PROGRAM OP70_CONVEYOR
VAR
	con_step_no : INT;
	cam_trig : BOOL;
	cam_ok : BOOL;
	LH_Cam_OK : BOOL;
	RH_Cam_OK : BOOL;
	t1: ton;
	t2: ton;
	t3: ton;
	t4: ton;
	
	temp: BOOL;
	check:BOOL;
	check1:ton;
	fwd_time : INT :=500;
	rev_time : INT :=500;	
	count_nok :INT;
	forward: BOOL;
	reverse: BOOL;

	temp1: BOOL;
	temp2: BOOL;
	
	LH_Cyl_Delay : TON;
	RH_Cyl_Delay : TON;
	temp_3: BOOL;
END_VAR

IF (NOT OP70_AutoSelected OR OP70_ErrorActive ) THEN
	//SR70_CONV_servo_ctrl.VELmove_Start:=FALSE;
	forward:=FALSE;
	reverse:=FALSE;
	con_step_no:= 10;
END_IF	



IF MANUAL_SELECTED AND OP70_ManualSelected THEN               
	IF I70_DRUM_CONV_REV_I308_3 THEN
		SR70_Conv_servo_status.targetVelocity:=OP70_Conv_Rev_Speed_6_3;
		SR70_CONV_servo_ctrl.VELmove_Start:=I70_DRUM_CONV_REV_I308_3;
 	ELSIF I70_DRUM_CONV_FWD_I308_4 THEN
		SR70_Conv_servo_status.targetVelocity:=OP70_Conv_Fwd_Speed_7_89;
		SR70_CONV_servo_ctrl.VELmove_Start:=I70_DRUM_CONV_FWD_I308_4;	
	ELSE 	
		SR70_CONV_servo_ctrl.VELmove_Start:=0;   	
	END_IF  	
END_IF
                


CASE con_step_no OF
		10: IF (OP70_AutoSelected) THEN		// Check Automode Selected
				con_step_no:=65;
	        END_IF
		   
        65:	forward:=TRUE;
			SR70_CONV_servo_ctrl.Velocity:= OP70_Conveyor_Speed;
			SR70_CONV_servo_ctrl.VELmove_Start:=TRUE;	
			IF t2.Q THEN
    			forward:=FALSE;
				SR70_CONV_servo_ctrl.VELmove_Start:=FALSE;
				con_step_no:= 70;
			END_IF
		  
		70: IF NOT SR70_CONV_servo_ctrl.VELmove_Start THEN
			  cam_trig :=TRUE;
			  IF t1.Q THEN
				con_step_no:= 75;
			  END_IF
			END_IF	
					
		75:	IF cam_ok AND NOT SR70_CONV_servo_ctrl.VELmove_Start AND SR70_CONV_servo_ctrl.Axis_ready THEN
				IF LH_Cam_OK AND RH_Cam_OK THEN
				 con_step_no:= 90;
				 fwd_time:=OP70_Conv_Fwd_Time_6_3;
				 count_nok:=0;	
				ELSIF (NOT LH_Cam_OK OR NOT RH_Cam_OK) AND count_nok<5 THEN
				 count_nok := count_nok +1;
				 con_step_no:= 76;	
				ELSIF count_nok>=5 THEN
	             fwd_time:=7000;
				 con_step_no:= 80; 
				END_IF
			END_IF	
			
		76:	 IF NOT LH_Cam_OK AND NOT SR70_CONV_servo_ctrl.VELmove_Start THEN
				CR70_LH_Rej_Cyl.AutoCmd1:=0;
				CR70_LH_Rej_Cyl.AutoCmd2:=TRUE;
				con_step_no:= 78;
			ELSIF LH_Cam_OK THEN
				con_step_no:= 77;
			END_IF	
			
	   78:	IF I70_LH_REJ_CYL_REV_I1110_5 AND LH_Cyl_Delay.Q THEN
				CR70_LH_Rej_Cyl.AutoCmd1:=1;
				CR70_LH_Rej_Cyl.AutoCmd2:=0;
				con_step_no:= 79;					
			END_IF
			
	   79: IF I70_LH_REJ_CYL_FWD_I1110_4 AND count_nok<5 AND NOT CR70_LH_Rej_Cyl.AutoCmd2 THEN
				CR70_LH_Rej_Cyl.AutoCmd1:=0;
				con_step_no:= 77;
		   END_IF
           IF count_nok>5 THEN
			 fwd_time:=7000;
		     con_step_no:= 77;	
		   END_IF

			
	   77:	IF NOT RH_Cam_OK AND NOT SR70_CONV_servo_ctrl.VELmove_Start THEN	
				CR70_RH_Rej_Cyl.AutoCmd1:=0;
				CR70_RH_Rej_Cyl.AutoCmd2:=TRUE;				
				con_step_no:= 81;
			ELSIF RH_Cam_OK THEN
				con_step_no:= 80;
			END_IF

		81:	    IF  I70_RH_REJ_CYL_REV_I1110_7 AND RH_Cyl_Delay.Q THEN
					CR70_RH_Rej_Cyl.AutoCmd1:=1;
					CR70_RH_Rej_Cyl.AutoCmd2:=0;	
					con_step_no:= 82;			
				END_IF		
				
		82: 	IF I70_RH_REJ_CYL_FWD_I1110_6 AND count_nok<5 AND NOT CR70_RH_Rej_Cyl.AutoCmd2 THEN
					CR70_RH_Rej_Cyl.AutoCmd1:=0;					
					//fwd_time:=OP70_Conv_Fwd_Time_6_3;			  
				END_IF
				IF count_nok>5 THEN
					fwd_time:=7000;
				    con_step_no:= 80;	
				END_IF
	
		80: 	IF fwd_time=7000 THEN
			       count_nok:=0;	
				END_IF
                SR70_CONV_servo_ctrl.Velocity:= OP70_Conveyor_Speed;				
				forward:=TRUE;
				SR70_CONV_servo_ctrl.VELmove_Start:=TRUE;
				IF t2.Q THEN
    				forward:=FALSE;
					con_step_no:= 70;
					SR70_CONV_servo_ctrl.VELmove_Start:=FALSE;				
				END_IF
		        
		90: 	SR70_CONV_servo_ctrl.Velocity:= OP70_Conveyor_Speed;
				reverse:=TRUE;
				SR70_CONV_servo_ctrl.VELmove_Start:=TRUE;	
				IF t3.Q THEN				
 					reverse:=FALSE;
					SR70_CONV_servo_ctrl.VELmove_Start:=FALSE;
					con_step_no:= 100;				
				END_IF		
				
		100: OP70_pick_ready:=TRUE;
			 IF OP70_pick_done OR temp_3 THEN
				 OP70_pick_ready :=FALSE;
				 OP70_pick_done:=FALSE;
				 con_step_no:= 80;
			 END_IF
			 		
				
END_CASE

t1(IN:=cam_trig ,PT:=T#700MS);
IF cam_trig AND con_step_no=70  THEN // Reset for next cycle
	cam_ok:=FALSE;
	LH_Cam_OK:=0;
	RH_Cam_OK:=0;
END_IF

IF t1.Q THEN //Result updating from Camera
	cam_ok:=TRUE;
	LH_Cam_OK:=temp1;
	RH_Cam_OK:=temp2;
	cam_trig :=FALSE;
END_IF


t2(IN:=forward ,PT:=INT_TO_TIME(fwd_time));
t3(IN:=reverse ,PT:=INT_TO_TIME(rev_time));
t4(IN:=cam_ok,PT:=T#1S);

LH_Cyl_Delay(IN:= I70_LH_REJ_CYL_FWD_I1110_4 ,PT:=T#300MS);
RH_Cyl_Delay(IN:= I70_RH_REJ_CYL_FWD_I1110_6 ,PT:=T#300MS);

END_PROGRAM

(* stored: Version 1.1.0.1, ProductVersion 3.1.4024.11
   POU OP70_CONVEYOR: Id {e852cb9d-e89e-49d4-9fc2-04b9e9f18d93}, SpecialFunc None *)
